{attribute 'analysis' := '-33'}
TYPE ReadTest :
STRUCT
	ReadDynamicReadsAStructure					: DUT_TestStruct;
	ReadDynamicReadsAStructureAsync				: DUT_TestStruct;

	ReadGenericReturnsTheRequestedType			: ReadTestData;
	ReadGenericReturnsTheRequestedTypeAsync		: ReadTestData;
	
	ReadMultipleItemsInOneTransaction			: ReadTestData;
	ReadMultipleItemsInOneTransactionAsync		: ReadTestData;
	
	ReadValueReturnsTheExpectedValue			: ReadTestData;
	ReadValueReturnsTheExpectedValueAsync		: ReadTestData;
	
	WaitForValueThrowsExceptionOnTimeout		: BOOL;
	WaitForValueThrowsExceptionOnTimeoutAsync	: BOOL;
	
	WaitsForValueToChange						: ReadTestData;
	WaitsForValueToChangeAsync					: ReadTestData;
END_STRUCT
END_TYPE

(* stored: Version 1.1.0.1, ProductVersion 3.1.4024.12
   DUT ReadTest: Id {fce6c51c-6dfb-4a14-ae38-df59614254bd} *)
